# EPICS StreamDevice protocol: pnan5221/Db/pnan5221.proto
# pnan5221.proto for N5221 PNA Network Analyzer
Terminator = LF;

get_id {
   ReplyTimeout = 5000;
   out "*idn?";
   in "%#s";
}

sel_trace {
   out "calc:par:mnum \$1,fast";
}

get_freq {
   out "calc:par:mnum \$1,fast";
   out "calc:mark:x?";
   in "%f";
}

get_trace {
   Separator = ",";
   out "calc:par:mnum \$1,fast";
   out "calc:data? fdata";
   in "%f";
}

get_ampl_and_phase {
   out "calc:par:mnum \$1,fast";
   out "calc:mark:y?";
   in "%f,%(\$2)f";
}
